// TIA Portal project "Clase2Sim" (V14)

(* hardware
DEVICE "S71500/ET200MP station_1"  S7-1500 station
   slot 0: "Rail_0"  Rack  6ES7 590-1***0-0AA0
   slot 1: "Limon 1516"  CPU 1516F-3 PN/DP  6ES7 516-3FN01-0AB0  V2.1
      slot 3: "CPU display_1"  6ES7591-1BA00-0AA0
   slot 2: "DI 32x24VDC HF_1"  DI 32x24VDC HF  6ES7 521-1BL00-0AB0  V2.1
   slot 3: "DQ 32x24VDC/0.5A HF_1"  DQ 32x24VDC/0.5A HF  6ES7 522-1BL01-0AB0  V1.0
*)

// ===== PLC "Limon 1516"  CPU 1516F-3 PN/DP =====

VAR_GLOBAL   // PLC tag table "Default tag table"
   ""start"" AT %I0.0 : Bool;
   ""stop"" AT %I0.1 : Bool;
   ""L1"" AT %Q0.0 : Bool;
   ""L2"" AT %Q0.1 : Bool;
END_VAR